PROGRAM MAIN
VAR

END_VAR

DataShift();
HMI();

IF GVL_HMI.bTest THEN
	Test();	
END_IF

END_PROGRAM

(* stored: Version 1.1.0.1
   POU MAIN: Id {22e7d931-b4d7-4bf3-9673-d7ddeeeaad53}, SpecialFunc None *)
